// TIA Portal V20 export
// export: Created 2026-07-10T11:12:28.4639482Z, ExportSetting WithDefaults, DisplayName Totally Integrated Automation Portal, DisplayVersion V20, DisplayName TIA Portal Openness, DisplayVersion V20, DisplayName TIA Portal Version Control Interface, DisplayVersion V20, DisplayName STEP 7 Professional, DisplayVersion V20, DisplayName STEP 7 Safety, DisplayVersion V20, DisplayName WinCC Basic/Comfort/Advanced, DisplayVersion V20, DisplayName WinCC Unified, DisplayVersion V20
FUNCTION_BLOCK "WeightHandler"   // FB20, SCL
{ S7_Optimized_Access := 'TRUE' }
VERSION : 0.1
// stored: AutoNumber true, IsIECCheckEnabled false, IsRetainMemResEnabled false, MemoryReserve 100, SetENOAutomatically false, UDAEnableTagReadback false
   VAR_INPUT
      ValueMin : Real;
      ValueMax : Real;
      OutputMin : Real;
      OutputMax : Real;
      ValueOffset : Real;
      Value : Real;
   END_VAR
   VAR_OUTPUT
      Output : Real;
      Error : Bool;
   END_VAR
   VAR
      ConvertedValue : Real;
      TON1 { S7_SetPoint := 'True'} : TON_TIME;
   END_VAR
BEGIN
   #Error := FALSE;



   #ConvertedValue := (#Value - #ValueMin) / (#ValueMax - #ValueMin) * (#OutputMax - #OutputMin) + #OutputMin;
   #Output := #ConvertedValue + #ValueOffset;

   #TON1(IN := #ConvertedValue < 0.1,
         PT := T#60s,
         Q => #Error);

   IF #Output < 0 THEN
       #Output := 0;
   END_IF;
END_FUNCTION_BLOCK
